# EPICS autosave request: KsApp/Db/Ks_settings.req
$(P)$(R)ExposureMode
$(P)$(R)Format
$(P)$(R)NikonTriggerMode
$(P)$(R)CaptureMode
$(P)$(R)SignalExposureEnd
$(P)$(R)TriggerReady
$(P)$(R)SignalDeviceCapture
$(P)$(R)ExposureOutput
$(P)$(R)ExposureBias
$(P)$(R)TriggerFrameCt
$(P)$(R)TriggerDelay
$(P)$(R)ROIX
$(P)$(R)ROIY
$(P)$(R)NikonFrameRate
$(P)$(R)MeteringMode
$(P)$(R)ExposureTimeLimit
$(P)$(R)GainLimit
$(P)$(R)Brightness
$(P)$(R)MeteringAreaLeft
$(P)$(R)MeteringAreaTop
$(P)$(R)MeteringAreaWidth
$(P)$(R)MeteringAreaHeight
